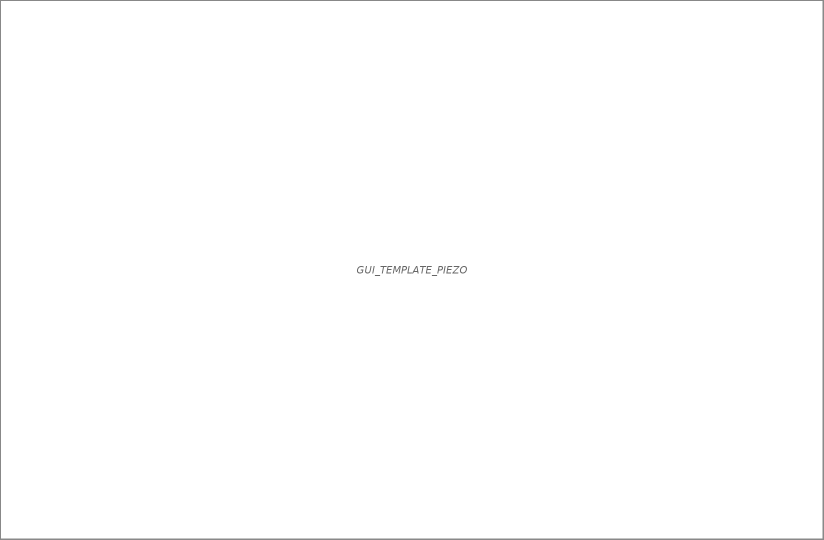
VISUALIZATION GUI_Piezo002  // 824x540
    Frame (0,0 824x540)
        shows GUI_TEMPLATE_PIEZO(m_Instance := MAIN.Piezo002)
END_VISUALIZATION

(* stored: Version 1.1.0.1, ProductVersion 3.1.4024.3
   Visu GUI_Piezo002: Id {34902cb3-70b9-49f0-b6c8-343ee5da4889} *)
